// TwinCAT 3 PLC project SPS
// ProgramVersion: 3.1.4026.10
// CompilerDefines: VISU_USEPROPERTYINFO
// libraries:
//   Tc2_ModbusRTU, * (Beckhoff Automation GmbH)
//   Tc2_SerialCom, * (Beckhoff Automation GmbH)
//   Tc2_Standard, * (Beckhoff Automation GmbH)
//   Tc2_System, * (Beckhoff Automation GmbH)
//   Tc2_TcpIp, * (Beckhoff Automation GmbH)
//   Tc2_Utilities, * (Beckhoff Automation GmbH)
//   VisuSymbols, 4.5.0.0 (System)
// project tree:
//   DUTs/01_Liste/01_Zustände/ ObjectState.TcDUT, SkillState.TcDUT (not stored), SystemState.TcDUT (not stored)
//   DUTs/01_Liste/02_Commands/ SkillCommand.TcDUT, SystemCommand.TcDUT
//   DUTs/01_Liste/03_Konfiguration/ Bewegungsart.TcDUT, Positionsart.TcDUT
//   DUTs/02_Schnittstellen/ I_State.TcIO
//   DUTs/03_Struktur/01_FB_Roboter/ PositionValues.TcDUT (not stored), Prozessvariablen.TcDUT (not stored), RealTimeData.TcDUT, ValueArray.TcDUT (not stored)
//   DUTs/03_Struktur/02_FB_Kraftsensor/ Kraftvariablen.TcDUT, Request.TcDUT (not stored), Response_Parameters.TcDUT (not stored), Response_Values.TcDUT (not stored)
//   DUTs/04_Union/ Array2Byte.TcDUT, Array4Byte.TcDUT, Array8Byte.TcDUT, INT2Byte.TcDUT, String2Byte.TcDUT
//   / GlobalTextList.TcGTLO, PlcTask.TcTTO, Visualization Manager.TcVMO (not stored)
//   GVLs/ GVL.TcGVL
//   POUs/01_Grundstruktur/ GrundstrukturObjekt.TcPOU
//   POUs/02_Objektklassen/ FB_Kraftsensor.TcPOU, FB_Roboter.TcPOU, FB_SmartGripper.TcPOU
//   POUs/ Anlage.TcPOU, MAIN.TcPOU, TestAblauf.TcPOU
//   VISUs/ Test.TcVIS
// real-time tasks:
//   TASK PlcTask: cycle T#10ms, priority 20, ADS port 350
//   TASK VISU_TASK: cycle T#200000us, priority 30, ADS port 351
// I/O:
//   DEVICE Gerät 1 (COM Port)
// variable links:
//   SPS/SPS Instance <-> Device 1 (COM Port)
//     PlcTask Inputs/GVL.Input/D[{0..63}] <-> Inputs/Data{1..64}  (64 links)
//     PlcTask Inputs/GVL.Input/SerStatus <-> Inputs/Status
//     PlcTask Outputs/Anlage.Gripper.Communication/OutData/D[{0..63}] <-> Outputs/Data{1..64}  (64 links)
//     PlcTask Outputs/Anlage.Gripper.Communication/OutData/SerCtrl <-> Outputs/Ctrl

CONFIGURATION SPS
    RESOURCE PLC ON TwinCAT3
        TASK PlcTask(INTERVAL := T#10ms, PRIORITY := 20);
        PROGRAM MAIN WITH PlcTask : MAIN;
    END_RESOURCE
END_CONFIGURATION

// ---- DUTs/01_Liste/01_Zustände/ObjectState.TcDUT
{attribute 'qualified_only'}
{attribute 'strict'}
{attribute 'to_string'}
TYPE ObjectState :
(
	AUS 			:= 0,				// Das Objekt ist ausgeschalten
	BEREIT 			:= 1,				// Das Objekt ist eingeschalten und bereit
	MANUELL			:= 2,				// Das Objekt befindet sich im Manuell-Modus
	LAUFEND 		:= 3,				// Das Objekt ist aktiv
	ABGESCHLOSSEN 	:= 4,				// Das Objekt hat den Prozess durchgeführt und hat selbständig gestoppt
	GESTOPPT 		:= 5,				// Das Objekt wurde gestoppt durch externe Einwirkung gestoppt
	FEHLER			:= 6				// Es gibt einen Fehler bezüglich des Objektes
);
END_TYPE

// ---- DUTs/01_Liste/02_Commands/SkillCommand.TcDUT
{attribute 'qualified_only'}
{attribute 'strict'}
{attribute 'to_string'}
TYPE SkillCommand :
(
	KEINE		:= 0,
	STARTEN		:= 1,
	STOPPEN		:= 2,
	RESETTEN 	:= 3
);
END_TYPE

// ---- DUTs/01_Liste/02_Commands/SystemCommand.TcDUT
{attribute 'qualified_only'}
{attribute 'strict'}
{attribute 'to_string'}
TYPE SystemCommand :
(
	KEINE		:= 0,
	AUSCHALTEN 	:= 1,
	EINSCHALTEN := 2,
	STOPPEN		:= 3,
	RESETTEN	:= 4
);
END_TYPE

// ---- DUTs/01_Liste/03_Konfiguration/Bewegungsart.TcDUT
{attribute 'qualified_only'}
{attribute 'strict'}
{attribute 'to_string'}
TYPE Bewegungsart :
(
	LinearToolSpace 			:= 0,		// Move to position (linear in tool-space)
	LinearJointSpace 			:= 1,		// Move to position (linear in joint-space)
	CircularToolSpace 			:= 2,		// Move Circular: Move to position (circular in tool-space)
	BlendCircularMoveLinear		:= 3		// Move Process
);
END_TYPE

// ---- DUTs/01_Liste/03_Konfiguration/Positionsart.TcDUT
{attribute 'qualified_only'}
{attribute 'strict'}
{attribute 'to_string'}
TYPE Positionsart :
(
	Absolut := 0,			// Absolute Bewegung bezogen auf Basis-Koordinatensystem
	Relativ := 1			// Relative Bewegung bezogen auf aktuelle Position
	
);
END_TYPE

// ---- DUTs/03_Struktur/01_FB_Roboter/RealTimeData.TcDUT
TYPE RealTimeData :
STRUCT
	messageSize 				: ARRAY[0..3] OF BYTE;
	timestamp 					: ARRAY[0..7] OF BYTE;
	//qTarget 					: ARRAY[0..47] OF BYTE;
	qTargetQ1 					: ARRAY[0..7] OF BYTE;
	qTargetQ2 					: ARRAY[0..7] OF BYTE;
	qTargetQ3 					: ARRAY[0..7] OF BYTE;
	qTargetQ4 					: ARRAY[0..7] OF BYTE;
	qTargetQ5 					: ARRAY[0..7] OF BYTE;
	qTargetQ6 					: ARRAY[0..7] OF BYTE;
	qdTarget 					: ARRAY[0..47] OF BYTE;
	qddTarget 					: ARRAY[0..47] OF BYTE;
	iTarget 					: ARRAY[0..47] OF BYTE;
	mTarget 					: ARRAY[0..47] OF BYTE;
	//qActual 					: ARRAY[0..47] OF BYTE;
	qActualQ1 					: ARRAY[0..7] OF BYTE;
	qActualQ2 					: ARRAY[0..7] OF BYTE;
	qActualQ3 					: ARRAY[0..7] OF BYTE;
	qActualQ4 					: ARRAY[0..7] OF BYTE;
	qActualQ5 					: ARRAY[0..7] OF BYTE;
	qActualQ6 					: ARRAY[0..7] OF BYTE;
	//qdActual 					: ARRAY[0..47] OF BYTE;
	qdActualQ1 					: ARRAY[0..7] OF BYTE;
	qdActualQ2 					: ARRAY[0..7] OF BYTE;
	qdActualQ3 					: ARRAY[0..7] OF BYTE;
	qdActualQ4 					: ARRAY[0..7] OF BYTE;
	qdActualQ5 					: ARRAY[0..7] OF BYTE;
	qdActualQ6 					: ARRAY[0..7] OF BYTE;
	iActual 					: ARRAY[0..47] OF BYTE;
	toolAccelerometerValues 	: ARRAY[0..23] OF BYTE;
	unused_1					: ARRAY[0..119] OF BYTE;
	tcpForce 					: ARRAY[0..47] OF BYTE;
	//toolVector 					: ARRAY[0..47] OF BYTE;
	toolVectorQ1 				: ARRAY[0..7] OF BYTE;
	toolVectorQ2 				: ARRAY[0..7] OF BYTE;
	toolVectorQ3 				: ARRAY[0..7] OF BYTE;
	toolVectorQ4 				: ARRAY[0..7] OF BYTE;
	toolVectorQ5 				: ARRAY[0..7] OF BYTE;
	toolVectorQ6 				: ARRAY[0..7] OF BYTE;
	tcpSpeed 					: ARRAY[0..47] OF BYTE;
	digitalInputBits 			: ARRAY[0..7] OF BYTE;
	unused_2					: ARRAY[0..119] OF BYTE;
END_STRUCT
END_TYPE

// ---- DUTs/03_Struktur/02_FB_Kraftsensor/Kraftvariablen.TcDUT
TYPE Kraftvariablen :
STRUCT
	Fx					:LREAL;							// Kraft in X-Richtung 
	Fy					:LREAL;							// Kraft in Y-Richtung 
	Fz					:LREAL;							// Kraft in Z-Richtung 
	Tx					:LREAL;							// Moment auf X-Achse 
	Ty					:LREAL;							// Moment auf Y-Achse 
	Tz					:LREAL;							// Moment auf Z-Achse 
END_STRUCT
END_TYPE

// ---- DUTs/04_Union/Array2Byte.TcDUT
TYPE Array2Byte :
UNION
	arrByte 		:ARRAY[0..1] OF BYTE;
	sValue			:INT; 
END_UNION
END_TYPE

// ---- DUTs/04_Union/Array4Byte.TcDUT
TYPE Array4Byte :
UNION
	arrByte			:ARRAY[0..3] OF BYTE;
	rValue			:INT;
END_UNION
END_TYPE

// ---- DUTs/04_Union/Array8Byte.TcDUT
TYPE Array8Byte :
UNION
	arrByte			:ARRAY[0..7] OF BYTE;
	rValue			:LREAL;
END_UNION
END_TYPE

// ---- DUTs/04_Union/INT2Byte.TcDUT
TYPE INT2Byte :
UNION
	sValue			:INT; 
	arrByte 		:ARRAY[0..1] OF BYTE;
END_UNION
END_TYPE

// ---- DUTs/04_Union/String2Byte.TcDUT
TYPE String2Byte :
UNION
	sValue			:STRING; 
	arrByte 		:ARRAY[0..255] OF BYTE;
END_UNION
END_TYPE

// ---- GVLs/GVL.TcGVL
{attribute 'qualified_only'}
VAR_GLOBAL
	Input				AT%I*	:PcComInData;
	Output				AT%Q*	:PcComOutData;
END_VAR

// ---- DUTs/02_Schnittstellen/I_State.TcIO
INTERFACE I_State

PROPERTY P_State : INT
GET
END_GET
END_PROPERTY

END_INTERFACE

// ---- POUs/MAIN.TcPOU
PROGRAM MAIN
VAR_INPUT
	SysCommand			:SystemCommand;
	SkillCommand		:Skillcommand;
	testProcessValue	:Prozessvariablen; 
	
	Switch				:BOOL;

	
END_VAR

Anlage();
TestAblauf();

END_PROGRAM

// ---- POUs/Anlage.TcPOU
PROGRAM Anlage
VAR
	UR5				:FB_Roboter;
	Gripper			:FB_SmartGripper;
	HEX_E			:FB_Kraftsensor; 
END_VAR

UR5(
    sIP := '192.168.50.100',
    iPort_Prim := 30002,
    iPort_RT := 30003,
    Prozessvariablen := MAIN.testProcessValue); // FB_Roboter
Gripper(); // FB_SmartGripper
HEX_E(
    iSkillCommand := MAIN.SkillCommand,
    iSysCommand := MAIN.SysCommand,
    sIP := '192.168.1.1',
    iPort := 49151); // FB_Kraftsensor

END_PROGRAM

// ---- POUs/02_Objektklassen/FB_Roboter.TcPOU
FUNCTION_BLOCK FB_Roboter EXTENDS GrundstrukturObjekt
VAR_INPUT
	// Kommunikationsvariablen
	sIP					:T_IPv4Addr;
	iPort_Prim			:UINT;
	iPort_RT			:UINT;
	
	// Prozessvariablen
	Prozessvariablen: 	Prozessvariablen;
END_VAR

VAR_OUTPUT
END_VAR

VAR
	// Instanziierung von Kommunikationsbausteine
	Connect				:FB_SocketConnect;
	Disconnect			:FB_SocketCloseALL;
	Send_START			:FB_SocketSend;
	Send_STOP			:FB_SocketSend;
	Connect_RT			:FB_SocketConnect;
	Receive_RT			:FB_SocketReceive;
	Disconnect_RT		:FB_SocketClose;
	
	// Kommunikationsvariablen
	sSrvNetId   		:T_AmsNetId := '';
	tTimeout    		:TIME := T#45S;(*!!!*)
	hSocket    			:T_HSOCKET;
	hSocket_RT    		:T_HSOCKET;
	
	// Managementvariablen
	Connect_State		:BOOL;
	Disconnect_State	:BOOL;
	bTurnedOn 			:BOOL;
	
	bVerbinden			:BOOL;
	bTrennen			:BOOL;
	bBewegungZuPosition	:BOOL;
	bBewegungStoppen	:BOOL;
	
	Delay_1				:TON;
	Delay_2				:TON;
	
	bQ1					:BOOL;
	bQ2					:BOOL;
	bQ3					:BOOL;
	bQ4					:BOOL;
	bQ5					:BOOL;
	bQ6					:BOOL;
	
	// RealTimeDatenerfassung
	RT_State			:INT;							// RealTime-State-Variable
	ReceivedData		:RealTimedata;					// Erhaltene Daten von Roboter
	nRecBytes			:UDINT;							// Anzahl der erhaltenen Bytes
	
	JointPositions		:PositionValues;				// Ausgelesene aktuelle Joint-Positonen-Byte
	JointSpeed			:PositionValues;				// Ausgelesene aktuelle Joint-Geschwindigkeit-Byte
	ToolPosition		:PositionValues;				// Ausgelesene aktuelle Tool-Positonen-Byte
	
	TempJointPosRev		:ValueArray;					// Ausgelesene aktuelle Joint-Positonen-Byte (Reversed)
	TempJointVRev		:valueArray;					// Ausgelesene aktuelle Joint-Geschwindigkeit-Byte (Reversed)	
	TempToolPosRev		:ValueArray;					// Ausgelesene aktuelle Tool-Positonen-Byte(Reversed)
	
	Joint				:Array8Byte;					// Aktuelle Joint-Positonen
	JSpeed				:Array8Byte;					// Aktuelle Joint-Geschwindgeit
	Tool				:Array8Byte;					// Aktuelle Tool-Positionen
	m					:INT;							// Loop-Variable
	
	// Prozessdaten
	TargetPosition		:Positionvalues;				// Targetpositions
	bSetValues			:BOOL;

END_VAR

// Instanziierungen
	Connect_RT(sSrvNetId := sSrvNetId,
							sRemoteHost := sIP,
							nRemotePort := iPort_RT,
							tTimeout := tTimeout,
							bBusy => bBusy,
							bError => bError,
							nErrId => iErrorID,
							hSocket => hSocket_RT);	
							
	Send_START(sSrvNetId := sSrvNetId,
			hSocket := hSocket,
			tTimeout := tTimeout,
			bBusy => bBusy,
			bError => bError,
			nErrId => iErrorID);
	Send_STOP(sSrvNetId := sSrvNetId,
			hSocket := hSocket,
			tTimeout := tTimeout,
			bBusy => bBusy,
			bError => bError,
			nErrId => iErrorID);
							
	Receive_RT(sSrvNetId := sSrvNetId,
							hSocket := hSocket_RT,
							cbLen := SIZEOF(ReceivedData),
							pDest := ADR(ReceivedData),
							tTimeout := tTimeout,
							bBusy => bBusy,
							bError => bError,
							nErrId => iErrorID,
							nRecBytes => nRecBytes);
							
	Disconnect_RT(sSrvNetId := sSrvNetId,
							hSocket := hSocket_RT,
							tTimeout := tTimeout,
							bBusy => bBusy,
							bError => bError,
							nErrId => iErrorID);

//____________________________________________________________________________________________
// Input-Command-Verwaltung
IF iSysCommand = 2 AND iState = 0 THEN			// System schaltet Objekt ein
	Connect_State := TRUE;
END_IF

IF iSysCommand = 1 AND iState = 1 THEN			// System schaltet Objekt aus
	Disconnect_State := TRUE;				
END_IF
//____________________________________________________________________________________________
// Interner Methodenaufruf (Durch System oder Skill)
IF Connect_State THEN
	bVerbinden := Verbinden();
	bTurnedOn := TRUE;
END_IF

IF Disconnect_State THEN
	bTrennen := Trennen();
	bTurnedOn := FALSE;;
END_IF

//____________________________________________________________________________________________
// Datenerfassungsprozess
IF bTurnedOn THEN
	CASE RT_State OF 
		0:	// Connect to RealTimePort
				Connect_RT(bExecute := TRUE);			
					
				IF NOT Connect_RT.bBusy AND NOT Connect_RT.bError THEN
					Connect_RT.bExecute := FALSE;
					RT_State := 1;
				END_IF
		
		1:	// Get Data 
				Receive_RT(bExecute := TRUE);
			
				IF NOT Receive_RT.bBusy AND NOT Receive_RT.bError THEN
					Receive_RT.bExecute := FALSE;
					RT_State := 2;
				END_IF
				
		2:	// Use Data
				m := 0;
		
				// Reverse Array
				FOR m := 0 TO 7 DO
					TempJointPosRev.q1[m] := ReceivedData.qActualQ1[7 - m];
					TempJointPosRev.q2[m] := ReceivedData.qActualQ2[7 - m];
					TempJointPosRev.q3[m] := ReceivedData.qActualQ3[7 - m];
					TempJointPosRev.q4[m] := ReceivedData.qActualQ4[7 - m];
					TempJointPosRev.q5[m] := ReceivedData.qActualQ5[7 - m];
					TempJointPosRev.q6[m] := ReceivedData.qActualQ6[7 - m];
					
					TempJointVRev.q1[m] := ReceivedData.qdActualQ1[7 - m];
					TempJointVRev.q2[m] := ReceivedData.qdActualQ2[7 - m];
					TempJointVRev.q3[m] := ReceivedData.qdActualQ3[7 - m];
					TempJointVRev.q4[m] := ReceivedData.qdActualQ4[7 - m];
					TempJointVRev.q5[m] := ReceivedData.qdActualQ5[7 - m];
					TempJointVRev.q6[m] := ReceivedData.qdActualQ6[7 - m];
					
					TempToolPosRev.q1[m] := ReceivedData.toolVectorQ1[7 - m];
					TempToolPosRev.q2[m] := ReceivedData.toolVectorQ2[7 - m];
					TempToolPosRev.q3[m] := ReceivedData.toolVectorQ3[7 - m];
					TempToolPosRev.q4[m] := ReceivedData.toolVectorQ4[7 - m];
					TempToolPosRev.q5[m] := ReceivedData.toolVectorQ5[7 - m];
					TempToolPosRev.q6[m] := ReceivedData.toolVectorQ6[7 - m];
				END_FOR
			
				Joint.arrByte := TempJointPosRev.q1;
				JointPositions.q1 := RAD_TO_DEG(Joint.rValue);
				Joint.arrByte := TempJointPosRev.q2;
				JointPositions.q2 := RAD_TO_DEG(Joint.rValue);
				Joint.arrByte := TempJointPosRev.q3;
				JointPositions.q3 := RAD_TO_DEG(Joint.rValue);
				Joint.arrByte := TempJointPosRev.q4;
				JointPositions.q4 := RAD_TO_DEG(Joint.rValue);
				Joint.arrByte := TempJointPosRev.q5;
				JointPositions.q5 := RAD_TO_DEG(Joint.rValue);
				Joint.arrByte := TempJointPosRev.q6;
				JointPositions.q6 := RAD_TO_DEG(Joint.rValue);
				
				JSpeed.arrByte := TempJointVRev.q1;
				JointSpeed.q1 := JSpeed.rValue;
				JSpeed.arrByte := TempJointVRev.q2;
				JointSpeed.q2 := JSpeed.rValue;
				JSpeed.arrByte := TempJointVRev.q3;
				JointSpeed.q3 := JSpeed.rValue;
				JSpeed.arrByte := TempJointVRev.q4;
				JointSpeed.q4 := JSpeed.rValue;
				JSpeed.arrByte := TempJointVRev.q5;
				JointSpeed.q5 := JSpeed.rValue;
				JSpeed.arrByte := TempJointVRev.q6;
				JointSpeed.q6 := JSpeed.rValue;
				
				Tool.arrByte := TempToolPosRev.q1;
				ToolPosition.q1 := Tool.rValue;
				Tool.arrByte := TempToolPosRev.q2;
				ToolPosition.q2 := Tool.rValue;
				Tool.arrByte := TempToolPosRev.q3;
				ToolPosition.q3 := Tool.rValue;
				Tool.arrByte := TempToolPosRev.q4;
				ToolPosition.q4 := RAD_TO_DEG(Tool.rValue);
				Tool.arrByte := TempToolPosRev.q5;
				ToolPosition.q5 := RAD_TO_DEG(Tool.rValue);
				Tool.arrByte := TempToolPosRev.q6;
				ToolPosition.q6 := RAD_TO_DEG(Tool.rValue);
				
				Delay_2(IN := TRUE, PT := T#0.5S);
				IF Delay_2.Q THEN
					Delay_2(IN := FALSE);
					RT_State := 3;
				END_IF
				
		3:	// Disconnect from RealTimePort
				Disconnect_RT(bExecute := TRUE);
							
				IF NOT Disconnect_RT.bBusy AND NOT Disconnect_RT.bError THEN
					Disconnect_RT.bExecute := FALSE;
					RT_State := 0;
				END_IF
		
	END_CASE
END_IF
//____________________________________________________________________________________________
// Zustandsmanagement

IF bError THEN 
	iState := 6;
END_IF

CASE iState OF 
	0: // AUS
		// DO
		
		// TRANSITION
			IF bVerbinden THEN							// Verbindung wird aufgebaut
				Connect_State := FALSE;
				bVerbinden := FALSE;
				iState := 1;
			END_IF
			
	//____________________________________________________________________________________________
	1: // BEREIT
		// DO
			IF iSkillCommand = 1 THEN
				bBewegungZuPosition := A_BewegungZuPosition();
			END_IF
			
			IF bBewegungZuPosition THEN
				Delay_1(IN := TRUE, PT := T#0.2S);
			END_IF
		
		// TRANSITION
			IF bTrennen THEN							// Verbindung wird getrennt
				Disconnect_State := FALSE;
				bTrennen := FALSE;
				iState := 0;
			END_IF
			
														// Manuell-Modus wird eingeschalten
													
			 IF Delay_1.Q THEN							// Objekt führt Prozessdurch
				 Delay_1(IN := FALSE);
				 bBewegungZuPosition := FALSE;
				 iState := 3;
			 END_IF			
	
	//____________________________________________________________________________________________
	2: // MANUELL
		// DO
		
		// TRANSITION
	
	//____________________________________________________________________________________________
	3: // LAUFEND
		// DO
			bBusy := TRUE;
			
			// Ermitteln von TargetPosition 
			IF NOT bSetvalues THEN
				// Kartesisch
				IF Prozessvariablen.MoveTyp = 0 THEN
					// Absolut
					IF Prozessvariablen.PosTyp = 0 THEN
						TargetPosition.q1 := Prozessvariablen.q1;
						TargetPosition.q2 := Prozessvariablen.q2;
						TargetPosition.q3 := Prozessvariablen.q3;
						TargetPosition.q4 := Prozessvariablen.q4;
						TargetPosition.q5 := Prozessvariablen.q5;
						TargetPosition.q6 := Prozessvariablen.q6;		
					END_IF
										
					// Relativ
					IF Prozessvariablen.PosTyp = 1 THEN
						TargetPosition.q1 := ToolPosition.q1 + Prozessvariablen.q1;
						TargetPosition.q2 := ToolPosition.q2 + Prozessvariablen.q2;
						TargetPosition.q3 := ToolPosition.q3 + Prozessvariablen.q3;
						TargetPosition.q4 := ToolPosition.q4 + Prozessvariablen.q4;
						TargetPosition.q5 := ToolPosition.q5 + Prozessvariablen.q5;
						TargetPosition.q6 := ToolPosition.q6 + Prozessvariablen.q6;
					END_IF
					
				END_IF
				
				// Gelenkwinkel
				IF Prozessvariablen.MoveTyp = 1 THEN
					TargetPosition.q1 := Prozessvariablen.q1;
					TargetPosition.q2 := Prozessvariablen.q2;
					TargetPosition.q3 := Prozessvariablen.q3;
					TargetPosition.q4 := Prozessvariablen.q4;
					TargetPosition.q5 := Prozessvariablen.q5;
					TargetPosition.q6 := Prozessvariablen.q6;	
				END_IF
			
				bSetvalues := TRUE;
			END_IF

			// Vergleich zwischen IST und SOLL
				// Kartesisch
				IF Prozessvariablen.MoveTyp = 0 THEN
					IF ABS(ABS(TargetPosition.q1) - ABS(ToolPosition.q1)) < 0.001 THEN
						bQ1 := TRUE;
					END_IF
					
					IF ABS(ABS(TargetPosition.q2) - ABS(ToolPosition.q2)) < 0.001 THEN
						bQ2 := TRUE;
					END_IF
					
					IF ABS(ABS(TargetPosition.q3) - ABS(ToolPosition.q3)) < 0.001 THEN
						bQ3 := TRUE;
					END_IF
					
					IF ABS(ABS(TargetPosition.q4) - ABS(ToolPosition.q4)) < 0.1 THEN
						bQ4 := TRUE;
					END_IF
					
					IF ABS(ABS(TargetPosition.q5) - ABS(ToolPosition.q5)) < 0.1 THEN
						bQ5 := TRUE;
					END_IF
					
					IF ABS(ABS(TargetPosition.q6) - ABS(ToolPosition.q6)) < 0.1 THEN
						bQ6 := TRUE;
					END_IF
				END_IF
				
				// Gelenkwinkel
				IF Prozessvariablen.MoveTyp = 1 THEN
					IF ABS(TargetPosition.q1) - ABS(JointPositions.q1) < 0.1 THEN
						bQ1 := TRUE;
					END_IF
					
					IF ABS(TargetPosition.q2) - ABS(JointPositions.q2) < 0.1 THEN
						bQ2 := TRUE;
					END_IF
					
					IF ABS(TargetPosition.q3) - ABS(JointPositions.q3) < 0.1 THEN
						bQ3 := TRUE;
					END_IF
					
					IF ABS(TargetPosition.q4) - ABS(JointPositions.q4) < 0.1 THEN
						bQ4 := TRUE;
					END_IF
					
					IF ABS(TargetPosition.q5) - ABS(JointPositions.q5) < 0.1 THEN
						bQ5 := TRUE;
					END_IF
					
					IF ABS(TargetPosition.q6) - ABS(JointPositions.q6) < 0.1 THEN
						bQ6 := TRUE;
					END_IF
				END_IF
			
		IF iSkillCommand = 2 OR iSysCommand = 3 THEN
			bBewegungStoppen := A_BewegungStoppen();
		END_IF
		
		// TRANSITION
			IF bQ1 AND bQ2 AND bQ3 AND bQ4 AND bQ5 AND bQ6 THEN									// Abgeschlossener Prozess
				bQ1 := FALSE;
				bQ2 := FALSE;
				bQ3 := FALSE;
				bQ4 := FALSE;
				bQ5 := FALSE;
				bQ6 := FALSE;
				
				bSetvalues := FALSE;
				bBusy := FALSE;
				iState := 4;
			END_IF
				
			IF bBewegungStoppen THEN
				bSetvalues := FALSE;																// Gestoppter Prozess
				bBusy := FALSE;
				iState := 5;
			END_IF
	
	//____________________________________________________________________________________________
	4: // ABGESCHLOSSEN
		// DO
			bDone := TRUE;
		
		// TRANSITION
			IF iSkillCommand = 3 OR iSysCommand = 4 THEN											// Objekt resetten											
				bDone := FALSE;
				iState := 1;
			END_IF
	//____________________________________________________________________________________________
	5: // GESTOPPT
		// DO
			IF iSkillCommand = 2 THEN																// Durch Skill beendet
				bDone := TRUE;
			END_IF
		
		// TRANSITION
			IF iSkillCommand = 3 OR iSysCommand = 4 THEN											// Objekt resetten
				bDone := FALSE;
				iState := 1;
			END_IF
	
	//____________________________________________________________________________________________
	6: // FEHLER
		// DO
			bDone := FALSE;
			bBusy := FALSE;
		
		// TRANSITION
			IF iSkillCommand = 3 OR iSysCommand = 3 THEN											// Objekt resetten
					iState := 1;
				END_IF
	
END_CASE

METHOD A_BewegungStoppen : BOOL
VAR_INPUT
END_VAR
VAR
	stringFormat   : FB_FormatString;		// Funktion für Stringerstellung	
	a				:INT := 2;

	Command			:T_MaxString;			// Commandstring
	CommandArray	:String2Byte;			// Byte-Array für Kommunikation mit Roboter
END_VAR
stringFormat(sFormat := 'stopj(%d)',
							arg1 := F_INT(a),
							bError => bError,
							nErrId => iErrorID,
							sOut => Command);	
							
// VOrbereiten von Array 
	CommandArray.sValue := Command;
	CommandArray.arrByte[LEN(CommandArray.sValue)] := 10;
	
// Senden von Array
	Send_STOP(cbLen := LEN(CommandArray.sValue),
			pSrc := ADR(CommandArray.arrByte),
			bExecute := TRUE);
			
	IF NOT bBusy THEN
		Send_STOP.bExecute := FALSE;
		A_BewegungStoppen := TRUE;
	END_IF
END_METHOD

METHOD A_BewegungZuPosition : BOOL
VAR 
	
	x					:LREAL;				// X-Koordinate
	y					:LREAL;				// Y-Koordinate
	z					:LREAL;				// Z-Koordinate
	rx					:LREAL;				// Orintierung um X-Achse
	ry					:LREAL;				// Orientierung um Y-Achse
	rz					:LREAL;				// Orientierung um Z-Achse
	
	q1					:LREAL;				// Joint-Position 1
	q2					:LREAL;				// Joint-Position 2
	q3					:LREAL;				// Joint-Position 3
	q4					:LREAL;				// Joint-Position 4
	q5					:LREAL;				// Joint-Position 5
	q6					:LREAL;				// Joint-Position 6

	stringFormat   : FB_FormatString;		// Funktion für Stringerstellung

	pose			:T_MaxString;			// Positionsstring
	Command			:T_MaxString;			// Commandstring
	
	CommandArray	:String2Byte;			// Byte-Array für Kommunikation mit Roboter
	
END_VAR
VAR_INPUT
	
END_VAR
// Einfluss von Positionart
	IF Prozessvariablen.PosTyp = 1 THEN		// Relative Bewegung
		
		x := ToolPosition.q1 + Prozessvariablen.q1;
		y := ToolPosition.q2 + Prozessvariablen.q2;
		z := ToolPosition.q3 + Prozessvariablen.q3;
		rx := DEG_TO_RAD(ToolPosition.q4 + Prozessvariablen.q4);
		ry := DEG_TO_RAD(ToolPosition.q5 + Prozessvariablen.q5);
		rz := DEG_TO_RAD(ToolPosition.q6 + Prozessvariablen.q6);
		
	END_IF
	
	IF Prozessvariablen.PosTyp = 0 THEN		// Absolute Bewegung
		
		x := Prozessvariablen.q1;
		y := Prozessvariablen.q2;
		z := Prozessvariablen.q3;
		rx := DEG_TO_RAD(Prozessvariablen.q4);
		ry := DEG_TO_RAD(Prozessvariablen.q5);
		rz := DEG_TO_RAD(Prozessvariablen.q6);
		
	END_IF
	
	stringFormat(sFormat := 'p[%.3f,%.3f,%.3f,%.3f,%.3f,%.3f]',
			arg1 := F_LREAL(x),
			arg2 := F_LREAL(y),
			arg3 := F_LREAL(z),
			arg4 := F_LREAL(rx),
			arg5 := F_LREAL(ry),
			arg6 := F_LREAL(rz),
			bError => bError,
			nErrId => iErrorID,
			sOut => pose);

// Einlfuss von Bewegungsart
	IF Prozessvariablen.MoveTyp = 0 THEN			// Move to position (linear in tool-space)
													// movel(pose, a=1.2, v=0.25, t=0, r=0)
		stringFormat(sFormat := 'movel(%s, a=%.2f, v=%.2f)',
							arg1 := F_STRING(pose),
							arg2 := F_LREAL(Prozessvariablen.a),
							arg3 := F_LREAL(Prozessvariablen.v),
							bError => bError,
							nErrId => iErrorID,
							sOut => Command);											
	END_IF
	
	IF Prozessvariablen.MoveTyp = 1 THEN			// Move to position (linear in joint-space)
													// movej(q, a=1.4, v=1.05, t=0, r =0)
		q1 := DEG_TO_RAD(Prozessvariablen.q4);
		q2 := DEG_TO_RAD(Prozessvariablen.q5);
		q3 := DEG_TO_RAD(Prozessvariablen.q6);
		q4 := DEG_TO_RAD(Prozessvariablen.q4);
		q5 := DEG_TO_RAD(Prozessvariablen.q5);
		q6 := DEG_TO_RAD(Prozessvariablen.q6);
		
		stringFormat(sFormat := 'movej([%.3f,%.3f,%.3f,%.3f,%.3f,%.3f], a=%.2f, v=%.2f)',
							arg1 := F_LREAL(q1),
							arg2 := F_LREAL(q2),
							arg3 := F_LREAL(q3),
							arg4 := F_LREAL(q4),
							arg5 := F_LREAL(q5),
							arg6 := F_LREAL(q6),
							arg7 := F_LREAL(Prozessvariablen.a),
							arg8 := F_LREAL(Prozessvariablen.v),
							bError => bError,
							nErrId => iErrorID,
							sOut => Command);	
													
	END_IF
	
	IF Prozessvariablen.MoveTyp = 2 THEN			// Move Circular: Move to position (circular in tool-space)
													//movec(pose_via, pose_to, a=1.2, v=0.25, r =0, mode=0)
													
		
	END_IF
	
	IF Prozessvariablen.MoveTyp = 3 THEN			// Move Process
													// movep(pose, a=1.2, v=0.25, r=0)
		stringFormat(sFormat := 'movep(%s, a=%.2f, v=%.2f)',
							arg1 := F_STRING(pose),
							arg2 := F_LREAL(Prozessvariablen.a),
							arg3 := F_LREAL(Prozessvariablen.v),
							bError => bError,
							nErrId => iErrorID,
							sOut => Command);												
	END_IF

// Vorbereiten von Array
	CommandArray.sValue := Command;
	CommandArray.arrByte[LEN(CommandArray.sValue)] := 10;

// Senden von Array	
	Send_START(cbLen := LEN(CommandArray.sValue),
			pSrc := ADR(CommandArray.arrByte),
			bExecute := TRUE);
			
	IF NOT bBusy THEN
		Send_START(bExecute := FALSE);
		A_BewegungZuPosition := TRUE;
	END_IF
END_METHOD

PROPERTY P_JointPosition : PositionValues
GET
P_JointPosition := JointPositions;
END_GET
END_PROPERTY

PROPERTY P_ToolPosition : PositionValues
GET
P_ToolPosition := ToolPosition;
END_GET
END_PROPERTY

METHOD Trennen : BOOL
VAR_INPUT
END_VAR
// Ausführen von Funktionalitäten
	Disconnect(sSrvNetId := sSrvNetId,
			bExecute := TRUE,
			tTimeout := tTimeout,
			bBusy => bBusy,
			bError => bError,
			nErrId => iErrorID);
	
	IF NOT bBusy AND NOT bError THEN
		Trennen := TRUE;
		Disconnect(bExecute := FALSE);
	END_IF
END_METHOD

METHOD Verbinden : BOOL 
VAR
	
END_VAR
// Ausführen von Funktionalitäten
	Connect(sSrvNetId := sSrvNetId,
			sRemoteHost := sIP,
			nRemotePort := iPort_Prim,
			bExecute := TRUE,
			tTimeout := tTimeout,
			bBusy => bBusy,
			bError => bError,
			nErrId => iErrorID,
			hSocket => hSocket);
			
	IF hSocket.handle <> 0 THEN
		Verbinden := TRUE;
		Connect(bExecute := FALSE);
		Connect_RT(bExecute := FALSE);
	END_IF
END_METHOD

END_FUNCTION_BLOCK

// ---- POUs/01_Grundstruktur/GrundstrukturObjekt.TcPOU
FUNCTION_BLOCK GrundstrukturObjekt IMPLEMENTS I_State
VAR_INPUT
	iMode				:INT;				// Information über aktuellen Betriebsmodi 
	iSkillCommand 		:SkillCommand;		// Steuerungsvariabel von Skill
	iSysCommand			:SystemCommand;		// Steuerungsvariabel von System
	iSysState			:SystemState;		// Information über Stand von System
END_VAR
VAR_OUTPUT
	bDone				:BOOL;				// Information ob Skill ausgfeührt wurde
	bBusy				:BOOL;				// Information ob Skill im Moment ausgeführt wird
	bError				:BOOL;				// Information ob sich Skill in Fehlerzustand befindet
	iErrorID			:UDINT;				// Information um welchen Fehler es sich handelt	
END_VAR
VAR
	iState				:ObjectState;		// Information über Zustand von Skill
END_VAR

PROPERTY P_State : INT
GET
P_State := iState;
END_GET
END_PROPERTY

END_FUNCTION_BLOCK

// ---- POUs/02_Objektklassen/FB_SmartGripper.TcPOU
FUNCTION_BLOCK FB_SmartGripper EXTENDS GrundstrukturObjekt
VAR_INPUT
	sIP					:T_IPv4Addr;
	iPort				:UINT;
END_VAR
VAR_OUTPUT
	
END_VAR
VAR
	// Instanziierung von Kommunikationsbausteine
	Communication		AT%Q*	:ModbusRtuMasterV2_PcCOM;
	

	
	// Kommunikationsvariablen
	UnitID      		:BYTE := 9;
    Quantity    		:WORD := 3;
    MBAddr      		:WORD := 1000;
    Execute_1     		:BOOL;
    Timeout     		:TIME := T#5S;
	
	cbRead				:UINT;

	Senddaten 			:ARRAY[0..2] OF INT;


END_VAR

// Instanziierungen
Senddaten[0] := 0;
Senddaten[1] := 0;
Senddaten[2] := 0;

//Communication_§end.WriteSingleRegister();
	Communication.WriteRegs(
		UnitID := UnitID,
		Quantity := Quantity,
		MBAddr := MBAddr,
		cbLength := SIZEOF(Senddaten),
		pMemoryAddr := ADR(Senddaten),
		Execute := Execute_1,
		Timeout := Timeout,
		BUSY => bBusy,
		Error => bError,
		ErrorId => iErrorID,
		cbRead => cbRead);
		
	//Communication.ReadRegs(
	//UnitID := UnitID,
	//Quantity := Quantity,
	//MBAddr := MBAddr,
	//cbLength := SIZEOF(Receivedaten),
	//pMemoryAddr := ADR(Receivedaten),
	//Execute := Execute_2,
	//Timeout := Timeout,
	//BUSY => bBusy,
	//Error => bError,
	//ErrorId => iErrorID,
	//cbRead => cbRead);
				

//____________________________________________________________________________________________
// Input-Command-Verwaltung

//____________________________________________________________________________________________
// Interner Methodenaufruf (Durch System oder Skill)

//____________________________________________________________________________________________
// Datenerfassungsprozess

//____________________________________________________________________________________________
// Zustandsmanagement

	CASE iState OF 
		0: // AUS
			// DO
		
			// TRANSITION
		
		//____________________________________________________________________________________________
		1: // BEREIT
			// DO

			// TRANSITION
		
		//____________________________________________________________________________________________
		2: // MANUELL
			// DO
		
			// TRANSITION
		
		//____________________________________________________________________________________________
		3: // LAUFEND
			// DO
		
			// TRANSITION
		
		//____________________________________________________________________________________________
		4: // ABGESCHLOSSEN
			// DO
		
			// TRANSITION
		
		//____________________________________________________________________________________________
		5: // GESTOPPT
			// DO
		
			// TRANSITION
		
		//____________________________________________________________________________________________
		6: // FEHLER
			// DO
		
			// TRANSITION
		
		
	END_CASE

METHOD DoSomething : BOOL
VAR_INPUT
	
END_VAR
VAR
	
END_VAR
END_METHOD

METHOD Trennen : BOOL
VAR_INPUT
END_VAR
END_METHOD

METHOD Verbinden : BOOL
VAR_INPUT
END_VAR
END_METHOD

END_FUNCTION_BLOCK

// ---- POUs/02_Objektklassen/FB_Kraftsensor.TcPOU
FUNCTION_BLOCK FB_Kraftsensor EXTENDS GrundstrukturObjekt
VAR_INPUT
	// Kommunikationsvariablen
	sIP					:T_IPv4Addr;
	iPort				:UINT;
END_VAR
VAR_OUTPUT
	
END_VAR
VAR
	// Instanziierung von Kommunikationsbausteine
	Connect				:FB_SocketConnect;
	Disconnect			:FB_SocketClose;
	Send				:FB_SocketSend;
	Receive				:FB_SocketReceive;
	
	// Kommunikationsvariablen
	sSrvNetId   		:T_AmsNetId := '';
	tTimeout    		:TIME := T#45S;(*!!!*)
	hSocket    			:T_HSOCKET;
	
	// RealTimeDatenerfassung
	RT_State			:INT;							// RealTime-State-Variable
	{attribute 'TcSwapWord'}
	SendData 			:Request;
	{attribute 'TcSwapWord'}
	ReceivedData		:Response_Values;				// Erhaltene Daten von Roboter
	nRecBytes			:UDINT;							// Anzahl der erhaltenen Bytes
	
	CPF					:INT := 10000;					// Counts per Force value
	CPT					:INT := 10000;					// Counts per Torque value (Noch mal 10 rechnen)
	ScalefactorFx		:INT := 200;					// Additional scaling factor (for the Fx,Fy,Fz,Tx,Ty,Tz)
	ScalefactorFy		:INT := 200;					// Additional scaling factor (for the Fx,Fy,Fz,Tx,Ty,Tz)
	ScalefactorFz		:INT := 200;					// Additional scaling factor (for the Fx,Fy,Fz,Tx,Ty,Tz)
	ScalefactorTx		:INT := 100;					// Additional scaling factor (for the Fx,Fy,Fz,Tx,Ty,Tz)
	ScalefactorTy		:INT := 100;					// Additional scaling factor (for the Fx,Fy,Fz,Tx,Ty,Tz)
	ScalefactorTz		:INT := 65;						// Additional scaling factor (for the Fx,Fy,Fz,Tx,Ty,Tz)
	
	RohArray			:INT2Byte;
	SwitchArray			:ARRAY[0..1] OF BYTE;
	SwichValue			:Array2Byte;
		
	Rohdaten			:Kraftvariablen;				// Rohwerte der Messung 
	Messung				:Kraftvariablen;				// Werte in Newton / Newtonmeter 

	// Managementvariablen
	bTurnedON			:BOOL;
	bStart				:BOOL;
	bStop				:BOOL;
	bReset				:BOOL;
	bManOn				:BOOL;
	m					:INT;
	
	// 
	
END_VAR

// Instanziierungen
Connect(sSrvNetId := sSrvNetId,
		sRemoteHost := sIP,
		nRemotePort := iPort,
		tTimeout := tTimeout,
		bBusy => bBusy,
		bError => bError,
		nErrId => iErrorID,
		hSocket => hSocket);	
						
Send(sSrvNetId := sSrvNetId,
		hSocket := hSocket,
		tTimeout := tTimeout,
		cbLen := SIZEOF(SendData),
		pSrc := ADR(SendData),
		bBusy => bBusy,
		bError => bError,
		nErrId => iErrorID);
						
Receive(sSrvNetId := sSrvNetId,
		hSocket := hSocket,
		cbLen := SIZEOF(ReceivedData),
		pDest := ADR(ReceivedData),
		tTimeout := tTimeout,
		bBusy => bBusy,
		bError => bError,
		nErrId => iErrorID,
		nRecBytes => nRecBytes);
						
Disconnect(sSrvNetId := sSrvNetId,
			hSocket := hSocket,
			tTimeout := tTimeout,
			bBusy => bBusy,
			bError => bError,
			nErrId => iErrorID);


//____________________________________________________________________________________________
// Input-Command-Verwaltung

//____________________________________________________________________________________________
// Interner Methodenaufruf (Durch System oder Skill)

//____________________________________________________________________________________________
// Datenerfassungsprozess
IF bManOn OR iState = 3 THEN
	CASE RT_State OF 
		0:	// Connect to RealTimePort
				Connect(bExecute := TRUE);			
					
				IF NOT Connect.bBusy AND NOT Connect.bError THEN
					Connect.bExecute := FALSE;
					RT_State := 1;
				END_IF
				
		1: 	// Send Data 
					SendData.Command := 0;
					Send(bExecute := TRUE);
				
					IF NOT Send.bBusy AND NOT Send.bError THEN
						Send.bExecute := FALSE;
						RT_State := 2;
					END_IF
		
		2:	// Get Data 
				Receive(bExecute := TRUE);
			
				IF NOT Receive.bBusy AND NOT Receive.bError THEN
					Receive.bExecute := FALSE;
					RT_State := 3;
				END_IF
				
		3:	// Convert Data
		
			RohArray.sValue := ReceivedData.Fx;
			SwitchArray[0] := RohArray.arrByte[1];
			SwitchArray[1] := RohArray.arrByte[0];
			SwichValue.arrByte := SwitchArray;
			Rohdaten.Fx := SwichValue.sValue;
			Messung.Fx := Rohdaten.Fx * ScalefactorFx / (CPF);
			
			RohArray.sValue := ReceivedData.Fy;
			SwitchArray[0] := RohArray.arrByte[1];
			SwitchArray[1] := RohArray.arrByte[0];
			SwichValue.arrByte := SwitchArray;
			Rohdaten.Fy := SwichValue.sValue;
			Messung.Fy := Rohdaten.Fy * ScalefactorFy / (CPF);
			
			RohArray.sValue := ReceivedData.Fz;
			SwitchArray[0] := RohArray.arrByte[1];
			SwitchArray[1] := RohArray.arrByte[0];
			SwichValue.arrByte := SwitchArray;
			Rohdaten.Fz := SwichValue.sValue;
			Messung.Fz := Rohdaten.Fz * ScalefactorFz / (CPF);
			
			RohArray.sValue := ReceivedData.Tx;
			SwitchArray[0] := RohArray.arrByte[1];
			SwitchArray[1] := RohArray.arrByte[0];
			SwichValue.arrByte := SwitchArray;
			Rohdaten.Tx := SwichValue.sValue;
			Messung.Tx := Rohdaten.Tx * ScalefactorTx / (CPT);
			
			RohArray.sValue := ReceivedData.Ty;
			SwitchArray[0] := RohArray.arrByte[1];
			SwitchArray[1] := RohArray.arrByte[0];
			SwichValue.arrByte := SwitchArray;
			Rohdaten.Ty := SwichValue.sValue;
			Messung.Ty := Rohdaten.Ty * ScalefactorTy / (CPT);
			
			RohArray.sValue := ReceivedData.Tz;
			SwitchArray[0] := RohArray.arrByte[1];
			SwitchArray[1] := RohArray.arrByte[0];
			SwichValue.arrByte := SwitchArray;
			Rohdaten.Tz := SwichValue.sValue;
			Messung.Tz := Rohdaten.Tz * ScalefactorTz / (CPT);
			
		
			RT_State := 4;
				
		4:	// Disconnect from RealTimePort
				Disconnect(bExecute := TRUE);
							
				IF NOT Disconnect.bBusy AND NOT Disconnect.bError THEN
					Disconnect.bExecute := FALSE;
					RT_State := 0;
				END_IF
		
	END_CASE
END_IF

//____________________________________________________________________________________________
// Zustandsmanagement

IF bError THEN 
	iState := 6;
END_IF

CASE iState OF 
	0: // AUS
		// DO
		IF iSysCommand = 2 THEN			// System schaltet Objekt ein
			bTurnedON := TRUE;
		END_IF
	
		// TRANSITION
		IF bTurnedON THEN			// System schaltet Objekt ein
			iState := 1;
		END_IF
	//____________________________________________________________________________________________
	1: // BEREIT
		// DO
		IF iSysCommand = 1 THEN																		// System schaltet Objekt aus
			bTurnedON := FALSE;				
		END_IF
		
		IF iSkillCommand = 1 THEN
			bStart := TRUE;
		END_IF
	
		// TRANSITION
		IF NOT bTurnedON THEN																		// Objekt ausschalten
			Disconnect(bExecute := TRUE);
								
			IF NOT Disconnect.bBusy AND NOT Disconnect.bError THEN
				Disconnect.bExecute := FALSE;
				iState := 0;
			END_IF
		END_IF
		
																									// Objekt in Manuell-Modus
																									
		IF bStart = 1 THEN	
			bStart := FALSE;																		// Objekt geht in Lauf-Modus
			iState := 3;
		END_IF																					
		
	
	//____________________________________________________________________________________________
	2: // MANUELL
		// DO
	
		// TRANSITION
	
	//____________________________________________________________________________________________
	3: // LAUFEND
		// DO
		bBusy := TRUE;
		
		IF iSkillCommand = 2 OR iSysCommand = 3 THEN	
			bStop := TRUE;
		END_IF
	
		// TRANSITION
		IF bStop  THEN																						// Objekt wird gestoppt durch Skill												
			IF RT_State = 0 THEN
				bStop := FALSE;
				iState := 5;
			END_IF
		END_IF
	
	//____________________________________________________________________________________________
	4: // ABGESCHLOSSEN
		// DO
	
		// TRANSITION
	
	//____________________________________________________________________________________________
	5: // GESTOPPT
		// DO
		bBusy := FALSE;
		bDone := TRUE;
		
		Messung.Fx := 0;
		Messung.Fy := 0;
		Messung.Fz := 0;
		Messung.Tx := 0;
		Messung.Ty := 0;
		Messung.Tz := 0;
		
		IF iSkillCommand = 3 OR iSysCommand = 4 THEN												// Befehl für Resetten wird gegeben
			bReset := TRUE;
		END_IF
	
		// TRANSITION
		IF bReset THEN
			bReset := FALSE;
			bDone := FALSE;
			iState := 1;
		END_IF
	
	//____________________________________________________________________________________________
	6: // FEHLER
		// DO
		bBusy := FALSE;
		
		Messung.Fx := 0;
		Messung.Fy := 0;
		Messung.Fz := 0;
		Messung.Tx := 0;
		Messung.Ty := 0;
		Messung.Tz := 0;
		
		IF iSkillCommand = 3 OR iSysCommand = 4 THEN												// Befehl für Resetten wird gegeben
			bReset := TRUE;
		END_IF
	
		// TRANSITION
		IF bReset THEN
			bError := FALSE;
			bReset := FALSE;
			bDone := FALSE;
			iState := 1;
		END_IF
	
	
END_CASE

PROPERTY P_Messdaten : Kraftvariablen
GET
P_Messdaten := Messung;
END_GET
END_PROPERTY

END_FUNCTION_BLOCK

// ---- POUs/TestAblauf.TcPOU
PROGRAM TestAblauf
VAR
END_VAR

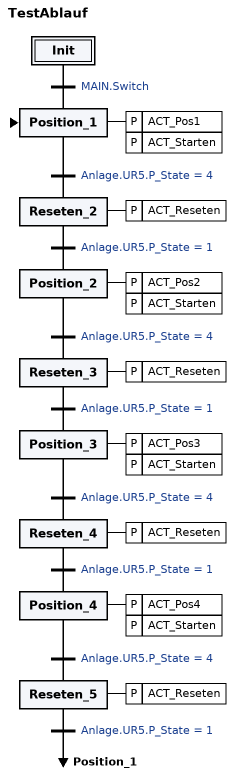
INITIAL_STEP Init:
END_STEP
TRANSITION FROM Init TO Position_1
    := MAIN.Switch;
END_TRANSITION
STEP Position_1:
    ACT_Pos1(P);
    ACT_Starten(P);
END_STEP
TRANSITION FROM Position_1 TO Reseten_2
    := Anlage.UR5.P_State = 4;
END_TRANSITION
STEP Reseten_2:
    ACT_Reseten(P);
END_STEP
TRANSITION FROM Reseten_2 TO Position_2
    := Anlage.UR5.P_State = 1;
END_TRANSITION
STEP Position_2:
    ACT_Pos2(P);
    ACT_Starten(P);
END_STEP
TRANSITION FROM Position_2 TO Reseten_3
    := Anlage.UR5.P_State = 4;
END_TRANSITION
STEP Reseten_3:
    ACT_Reseten(P);
END_STEP
TRANSITION FROM Reseten_3 TO Position_3
    := Anlage.UR5.P_State = 1;
END_TRANSITION
STEP Position_3:
    ACT_Pos3(P);
    ACT_Starten(P);
END_STEP
TRANSITION FROM Position_3 TO Reseten_4
    := Anlage.UR5.P_State = 4;
END_TRANSITION
STEP Reseten_4:
    ACT_Reseten(P);
END_STEP
TRANSITION FROM Reseten_4 TO Position_4
    := Anlage.UR5.P_State = 1;
END_TRANSITION
STEP Position_4:
    ACT_Pos4(P);
    ACT_Starten(P);
END_STEP
TRANSITION FROM Position_4 TO Reseten_5
    := Anlage.UR5.P_State = 4;
END_TRANSITION
STEP Reseten_5:
    ACT_Reseten(P);
END_STEP
TRANSITION FROM Reseten_5 TO Position_1
    := Anlage.UR5.P_State = 1;
END_TRANSITION

ACTION ACT_Pos1:
MAIN.testProcessValue.q1 := 0.2;
MAIN.testProcessValue.q2 := 0;
MAIN.testProcessValue.q3 := 0;
MAIN.testProcessValue.q4 := 0;
MAIN.testProcessValue.q5 := 0;
MAIN.testProcessValue.q6 := 0;
MAIN.testProcessValue.a := 0.2;
MAIN.testProcessValue.v := 0.2;
MAIN.testProcessValue.MoveTyp := 0;
MAIN.testProcessValue.PosTyp := 1;
END_ACTION

ACTION ACT_Pos2:
MAIN.testProcessValue.q1 := 0;
MAIN.testProcessValue.q2 := 0.2;
MAIN.testProcessValue.q3 := 0;
MAIN.testProcessValue.q4 := 0;
MAIN.testProcessValue.q5 := 0;
MAIN.testProcessValue.q6 := 0;
MAIN.testProcessValue.a := 0.2;
MAIN.testProcessValue.v := 0.2;
MAIN.testProcessValue.MoveTyp := 0;
MAIN.testProcessValue.PosTyp := 1;
END_ACTION

ACTION ACT_Pos3:
MAIN.testProcessValue.q1 := -0.2;
MAIN.testProcessValue.q2 := 0;
MAIN.testProcessValue.q3 := 0;
MAIN.testProcessValue.q4 := 0;
MAIN.testProcessValue.q5 := 0;
MAIN.testProcessValue.q6 := 0;
MAIN.testProcessValue.a := 0.2;
MAIN.testProcessValue.v := 0.2;
MAIN.testProcessValue.MoveTyp := 0;
MAIN.testProcessValue.PosTyp := 1;
END_ACTION

ACTION ACT_Pos4:
MAIN.testProcessValue.q1 := 0;
MAIN.testProcessValue.q2 := -0.2;
MAIN.testProcessValue.q3 := 0;
MAIN.testProcessValue.q4 := 0;
MAIN.testProcessValue.q5 := 0;
MAIN.testProcessValue.q6 := 0;
MAIN.testProcessValue.a := 0.2;
MAIN.testProcessValue.v := 0.2;
MAIN.testProcessValue.MoveTyp := 0;
MAIN.testProcessValue.PosTyp := 1;
END_ACTION

ACTION ACT_Reseten:
MAIN.SkillCommand := 3;
END_ACTION

ACTION ACT_Starten:
MAIN.SkillCommand := 1;
END_ACTION

END_PROGRAM

// ---- GlobalTextList.TcGTLO
TEXTLIST GlobalTextList
  372 = '%s'
  874 = 'AUSCHALTEN'
  997 = 'Befehl'
  724 = 'Daten lesen'
  697 = 'Do'
  468 = 'EINSCHALTEN'
  779 = 'Erhaltene Daten'
  166 = 'Erhaltene Daten:'
  764 = 'KEINE'
  32 = 'Länge von Array:'
  525 = 'Länge von Message'
  162 = 'Länge von Message:'
  303 = 'RESETTEN'
  707 = 'SkillCommand'
  955 = 'START'
  554 = 'STARTEN'
  68 = 'Stopp'
  351 = 'STOPPEN'
  785 = 'SystemCommand'
  320 = 'Test'
  1 = 'Verbinden'
END_TEXTLIST

// ---- VISUs/Test.TcVIS
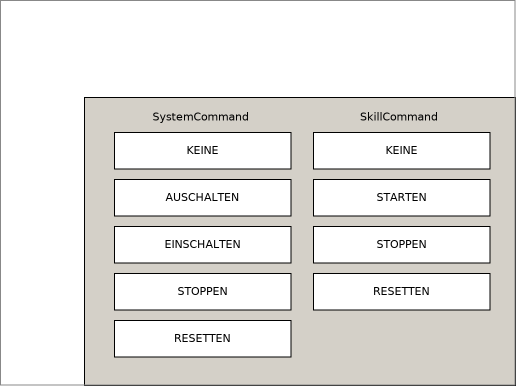
VISUALIZATION Test  // 516x386
    RoundedRectangle (84,97 432x289)
    RoundedRectangle (114,179 177x37), "AUSCHALTEN"
        OnMouseClick: execute { MAIN.SysCommand := 1; }
    RoundedRectangle (114,226 177x37), "EINSCHALTEN"
        OnMouseClick: execute { MAIN.SysCommand := 2; }
    RoundedRectangle (114,273 177x37), "STOPPEN"
        OnMouseClick: execute { MAIN.SysCommand := 3; }
    RoundedRectangle (114,320 177x37), "RESETTEN"
        OnMouseClick: execute { MAIN.SysCommand := 4; }
    RoundedRectangle (313,179 177x37), "STARTEN"
        OnMouseClick: execute { MAIN.SkillCommand := 1; }
    RoundedRectangle (313,226 177x37), "STOPPEN"
        OnMouseClick: execute { MAIN.SkillCommand := 2; }
    RoundedRectangle (313,273 177x37), "RESETTEN"
        OnMouseClick: execute { MAIN.SkillCommand := 3; }
    Label (126,102 150x30), "SystemCommand"
    Label (324,102 150x30), "SkillCommand"
    RoundedRectangle (114,132 177x37), "KEINE"
        OnMouseClick: execute { MAIN.SysCommand := 0; }
    RoundedRectangle (313,132 177x37), "KEINE"
        OnMouseClick: execute { MAIN.SkillCommand := 0; }
END_VISUALIZATION
